// TIA Portal V18 export
FUNCTION "AHUActualUnitStatesCtrl" : Void   // FC60105, LAD
{ S7_Optimized_Access := 'TRUE' }
VERSION : 0.1
// Operation Modes                                                 Unit State
// 0=Protection                                                         0=Stopped
// 1=Economy                                                           1=Checking-up  
// 2=PreComfort                                                       2=Preheating
// 3=Comfor                                                              3=Starting 
// 4=Auto(Scheduler)                                              4=RecirculatingOperation
//                                                                                 5=Economy Operation                                                                                                                                            6=PreComfort Operation 
//                                                                                 7=Comfort  operation
//                                                                                 8=Stopping
//                                                                                 9 =Blocking
// stored: AutoNumber false, IsIECCheckEnabled false, SetENOAutomatically false, UDAEnableTagReadback false
   VAR_INPUT
      iUnitID : Int;
      xManualSt1orSt2 : Bool;
      cTargetUnitState : Byte;
      cCheckingUpTime : Byte;
      cPreheatingTime : Byte;
      cStartingTime : Byte;
      cStoppingTime : Byte;
      cWorkOnFullRecycleTime : Byte;
   END_VAR
   VAR_OUTPUT
      cUnitStateForHMI : Byte;
   END_VAR
   VAR_IN_OUT
      cNextUnitState : Byte;
      xActualUnitStateEdge : Bool;
      cCounterToSwitchBtwStates : Int;
   END_VAR
   VAR_TEMP
      cState : Byte;
   END_VAR
BEGIN

REGION Network 1 (SCL)
   CASE #cTargetUnitState OF
       0:
           CASE #cNextUnitState OF
               0:  // 
                   IF #xActualUnitStateEdge THEN
                       #xActualUnitStateEdge := 0;
                   END_IF;
               1..7:  // 
                   #cNextUnitState := 8;
                   #xActualUnitStateEdge := 1;
                   ;
               8:
                   IF #xActualUnitStateEdge THEN
                       #xActualUnitStateEdge := 0;
                       IF #xManualSt1orSt2 THEN
                           #cCounterToSwitchBtwStates := 0;
                       ELSE
                           #cCounterToSwitchBtwStates := #cStoppingTime;
                       END_IF;
                   ELSIF #cCounterToSwitchBtwStates > 0 THEN
                       IF "Timer".x1SecRisingEdge THEN
                           #cCounterToSwitchBtwStates := #cCounterToSwitchBtwStates - 1;
                       END_IF;
                   ELSE
                       #cNextUnitState := 0;
                       #xActualUnitStateEdge := 1;
                   END_IF;
               9:
                   #cNextUnitState := 9;
           END_CASE;
       1..4:
           ;
       5..7:
           CASE #cNextUnitState OF
               0:  // 
                   #cNextUnitState := 1;
                   #xActualUnitStateEdge := 1;
               1:  // 
                   IF #xActualUnitStateEdge THEN
                       #xActualUnitStateEdge := 0;
                       IF #xManualSt1orSt2 THEN
                           #cCounterToSwitchBtwStates := 0;
                       ELSE
                           #cCounterToSwitchBtwStates := #cCheckingUpTime;
                       END_IF;

                   ELSIF #cCounterToSwitchBtwStates > 0 THEN
                       IF "Timer".x1SecRisingEdge THEN
                           #cCounterToSwitchBtwStates := #cCounterToSwitchBtwStates - 1;
                       END_IF;
                   ELSE
                       #cNextUnitState := 2;
                       #xActualUnitStateEdge := 1;
                   END_IF;
               2:
                   IF #xActualUnitStateEdge THEN
                       #xActualUnitStateEdge := 0;
                       IF #xManualSt1orSt2 OR "OAT".Temp.rOAT_Actual > "AHUFrostProt".FrostProt.OATtoStartPreheating[#iUnitID] THEN
                           // Statement section IF
                           #cCounterToSwitchBtwStates := 0;
                       ELSE
                           #cCounterToSwitchBtwStates := #cPreheatingTime;
                       END_IF;
                   ELSIF #cCounterToSwitchBtwStates > 0 THEN
                       IF "Timer".x1SecRisingEdge THEN
                           #cCounterToSwitchBtwStates := #cCounterToSwitchBtwStates - 1;
                       END_IF;
                   ELSE
                       #cNextUnitState := 3;
                       #xActualUnitStateEdge := 1;
                   END_IF;
               3:
                   IF #xActualUnitStateEdge THEN
                       #xActualUnitStateEdge := 0;
                       IF #xManualSt1orSt2 THEN
                           #cCounterToSwitchBtwStates := 0;
                       ELSE
                           #cCounterToSwitchBtwStates := #cStartingTime;
                       END_IF;

                   ELSIF #cCounterToSwitchBtwStates > 0 THEN
                       IF "Timer".x1SecRisingEdge THEN
                           #cCounterToSwitchBtwStates := #cCounterToSwitchBtwStates - 1;
                       END_IF;
                   ELSE
                       #cNextUnitState := 4;
                       #xActualUnitStateEdge := 1;
                   END_IF;
               4:
                   IF #xActualUnitStateEdge THEN
                       #xActualUnitStateEdge := 0;
                       #cCounterToSwitchBtwStates := #cWorkOnFullRecycleTime;
                   ELSIF #cCounterToSwitchBtwStates > 0 THEN
                       IF "Timer".x1SecRisingEdge THEN
                           #cCounterToSwitchBtwStates := #cCounterToSwitchBtwStates - 1;
                       END_IF;
                   ELSE
                       #cNextUnitState := #cTargetUnitState;  // transfer to Econom, PreComf, Comf
                       #xActualUnitStateEdge := 1;
                   END_IF;
               5..7:
                   IF #xActualUnitStateEdge THEN
                       #xActualUnitStateEdge := 0;
                   END_IF;
                   #cNextUnitState := #cTargetUnitState;
               8:
                   #cNextUnitState := 0;
               9:
                   #cNextUnitState := 9;
           END_CASE;
       8:
           ;
       9:
           #cNextUnitState := 9;
   END_CASE;
END_REGION

REGION Network 2 (SCL)
   IF "AHUEqp".Eqp.Cfg.cFan[#iUnitID] > 0 THEN
       IF #cNextUnitState > 2 AND #cNextUnitState < 9 THEN
           #cUnitStateForHMI := 2;
       ELSE
           #cUnitStateForHMI := 1;
       END_IF;
   ELSE
       #cUnitStateForHMI := 0;
   END_IF;
END_REGION
END_FUNCTION
